{attribute 'pack_mode' := '0'}
TYPE CyltronicProcessDataOutBytes :
STRUCT
	Byte0  : BYTE;
	Byte4  : BYTE;
	Byte3  : BYTE;
	Byte2  : BYTE;
	Byte1  : BYTE;
	Byte5  : BYTE;
	Byte6  : BYTE;
	Byte7  : BYTE;
END_STRUCT
END_TYPE

(* stored: Version 1.1.0.1, ProductVersion 3.1.4024.10
   DUT CyltronicProcessDataOutBytes: Id {9d689cae-ddb6-49d6-9c0f-09b2396bad33} *)
